(* CODESYS project Johnson,Joachim,Uppgift17.project

Project tree, tasks and I/O mapping:
  Device : CODESYS Control Win V3, 3S - Smart Software Solutions GmbH, order no. 305021, version 3.5.10.40
    application Application
      libraries: Standard, * (System)
      task MainTask (cyclic, interval t#20ms, priority 1) calls PLC_PRG, Lamp_Controll_Program [Controlling the lamp in the system], PrintoutAlarmCode
      program PLC_PRG [SFC]: MoveConv1to2, MoveCon2to3, Setrunning, SetStop, StopBTNCHECK, ResetAlarm, Convyor1to2Timout, Convyor2to3Timout
      global variables GVL
      Symbols
      program Lamp_Controll_Program [CFC]
      program Gui_Panel_Alarm [CFC]
      program PrintoutAlarmCode [CFC]
*)

// Device/Application/GVL
{attribute 'qualified_only'}
VAR_GLOBAL
	// signals from buttons
	iSUB00_S1: BOOL; // StartButton
	iSUB00_S2: BOOL; // Stopbutton
	iSUB00_S3: BOOL; // Resetbutton
	
	running: BOOL; 	// Is the aplication running
	alarm: BOOL; 	// Is the aplication running
	AlarmCode: word;
	
	// Signals from conveyors
	iSUB01_B1: BOOL; // Signals för conveyor 1. ontop
	iSUB02_B1: BOOL; // Signals för conveyor 2. ontop
	iSUB03_B1: BOOL; // Signals för conveyor 3. ontop
	
	// conveyor signal ontop conveyro.
	oSUB00_H1: BOOL; // Auto-On light
	oSUB00_H2: BOOL; // Alarm light
	oSUB00_H3: WORD; // Pallräknare
	
	// Motors
	oSUB01_K1: BOOL; // MOTOR FÖR converoyr 1
	oSUB02_K1: BOOL; // MOTOR FÖR converoyr 2
	oSUB03_K1: BOOL; // MOTOR FÖR converoyr 3
END_VAR

// Device/Application/PLC_PRG
PROGRAM PLC_PRG
VAR	
	TON_0: TON;
	OutputTime: TIME;
	TON2: TON;
	Output: TIME;
	TimeOutTimer: TON;
	TimeOutOutputTime: TIME;
	R_TRIG_0: R_TRIG;
	countercunt: CTD;
	countercunt3: CTD;
	countercunt4: CTD;
	Alarmcode: CTU;
	countercunt5: CTD;
END_VAR
VAR // added by the converter: edge detectors and wires of the graphical bodies
    _w1, _w3, _w5, _w6, _w12, _w14, _w15, _w17, _w19 : BOOL;
    _w2, _w4, _w7, _w8, _w9, _w10, _w11, _w13, _w16, _w18, _w20 : ANY;
END_VAR

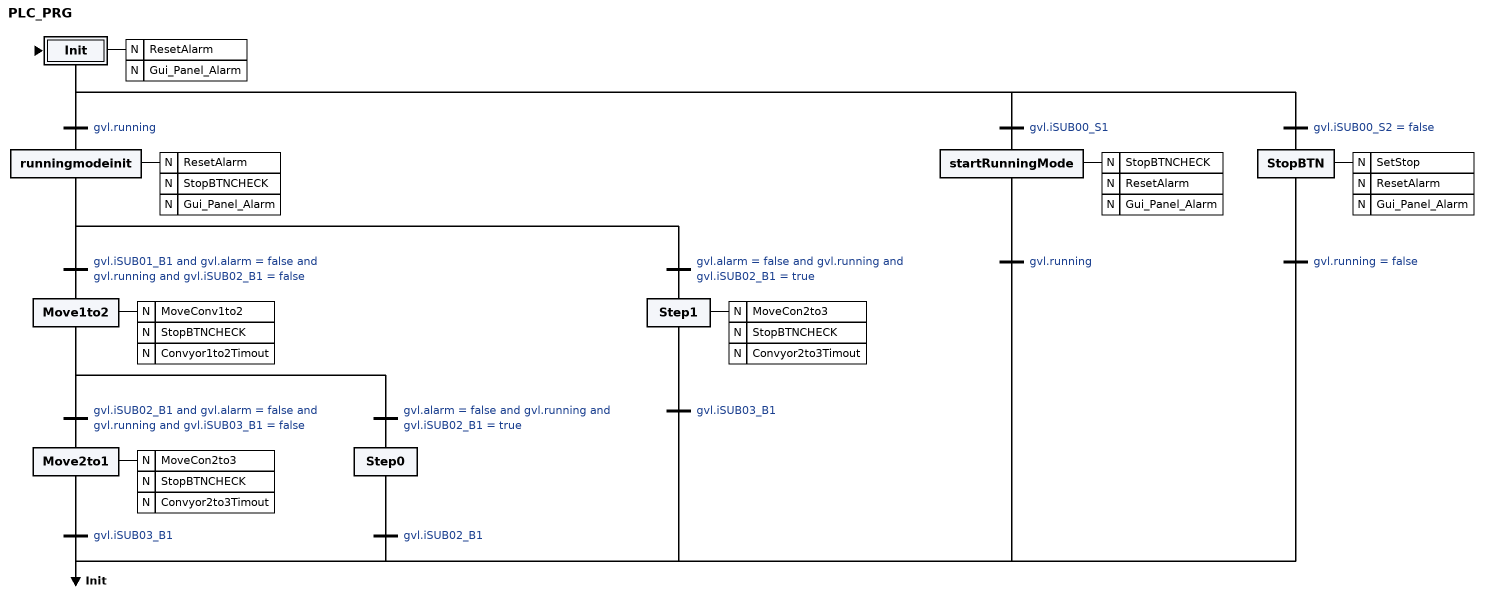
INITIAL_STEP Init:
    ResetAlarm(N);
    Gui_Panel_Alarm(N);
END_STEP
TRANSITION FROM Init TO runningmodeinit
    := gvl.running;
END_TRANSITION
STEP runningmodeinit:
    ResetAlarm(N);
    StopBTNCHECK(N);
    Gui_Panel_Alarm(N);
END_STEP
TRANSITION FROM runningmodeinit TO Move1to2
    := gvl.iSUB01_B1 and gvl.alarm = false and gvl.running and gvl.iSUB02_B1 = false;
END_TRANSITION
STEP Move1to2:
    MoveConv1to2(N);
    StopBTNCHECK(N);
    Convyor1to2Timout(N);
END_STEP
TRANSITION FROM Move1to2 TO Move2to1
    := gvl.iSUB02_B1 and gvl.alarm = false and gvl.running and gvl.iSUB03_B1 = false;
END_TRANSITION
STEP Move2to1:
    MoveCon2to3(N);
    StopBTNCHECK(N);
    Convyor2to3Timout(N);
END_STEP
TRANSITION FROM Move2to1 TO Init
    := gvl.iSUB03_B1;
END_TRANSITION
TRANSITION FROM Move1to2 TO Step0
    := gvl.alarm = false and gvl.running and gvl.iSUB02_B1 = true;
END_TRANSITION
STEP Step0:
END_STEP
TRANSITION FROM Step0 TO Init
    := gvl.iSUB02_B1;
END_TRANSITION
TRANSITION FROM runningmodeinit TO Step1
    := gvl.alarm = false and gvl.running and gvl.iSUB02_B1 = true;
END_TRANSITION
STEP Step1:
    MoveCon2to3(N);
    StopBTNCHECK(N);
    Convyor2to3Timout(N);
END_STEP
TRANSITION FROM Step1 TO Init
    := gvl.iSUB03_B1;
END_TRANSITION
TRANSITION FROM Init TO startRunningMode
    := gvl.iSUB00_S1;
END_TRANSITION
STEP startRunningMode:
    StopBTNCHECK(N);
    ResetAlarm(N);
    Gui_Panel_Alarm(N);
END_STEP
TRANSITION FROM startRunningMode TO Init
    := gvl.running;
END_TRANSITION
TRANSITION FROM Init TO StopBTN
    := gvl.iSUB00_S2 = false;
END_TRANSITION
STEP StopBTN:
    SetStop(N);
    ResetAlarm(N);
    Gui_Panel_Alarm(N);
END_STEP
TRANSITION FROM StopBTN TO Init
    := gvl.running = false;
END_TRANSITION

ACTION MoveConv1to2:
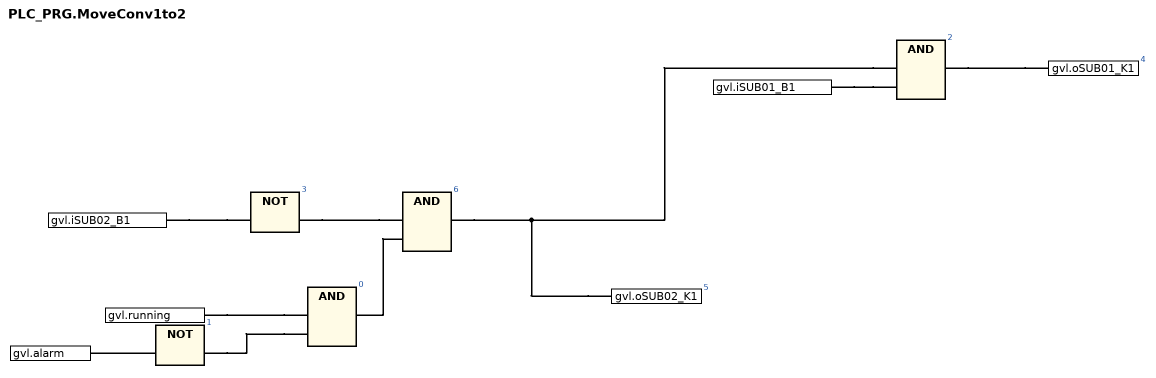
_w2 := gvl.running AND _w1;
_w1 := NOT gvl.alarm;
_w4 := NOT gvl.iSUB02_B1;
gvl.oSUB01_K1 := _w3 AND gvl.iSUB01_B1;
gvl.oSUB02_K1 := _w3;
_w3 := _w4 AND _w2;
END_ACTION

ACTION MoveCon2to3:
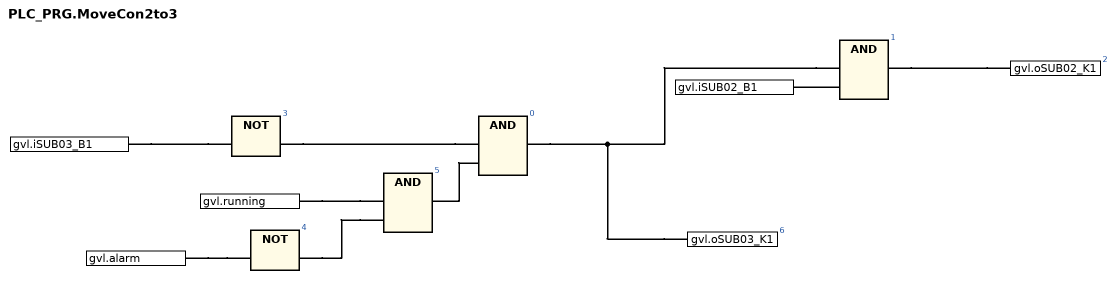
_w7 := _w5 AND _w6;
gvl.oSUB02_K1 := _w7 AND gvl.iSUB02_B1;
_w5 := NOT gvl.iSUB03_B1;
_w6 := gvl.running AND NOT gvl.alarm;
gvl.oSUB03_K1 := _w7;
END_ACTION

ACTION Setrunning:
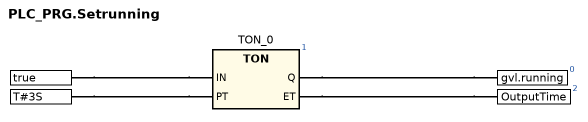
gvl.running := TON_0.Q;
TON_0(IN := true, PT := T#3S); // TON
OutputTime := TON_0.ET;
END_ACTION

ACTION SetStop:
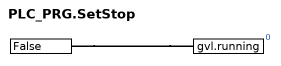
gvl.running := False;
END_ACTION

ACTION StopBTNCHECK:
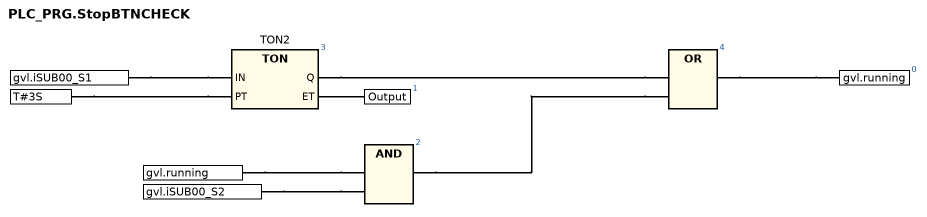
gvl.running := _w8;
Output := TON2.ET;
_w9 := gvl.running AND gvl.iSUB00_S2;
TON2(IN := gvl.iSUB00_S1, PT := T#3S); // TON
_w8 := TON2.Q OR _w9;
END_ACTION

ACTION ResetAlarm:
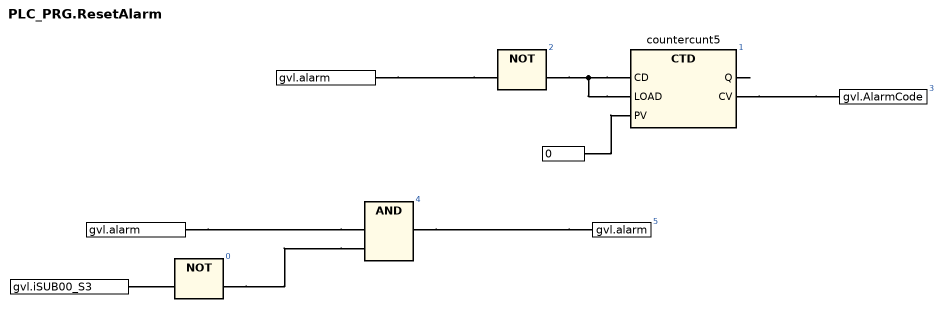
_w10 := NOT gvl.iSUB00_S3;
countercunt5(CD := _w11, LOAD := _w11, PV := 0); // CTD
_w11 := NOT gvl.alarm;
gvl.AlarmCode := countercunt5.CV;
gvl.alarm := gvl.alarm AND _w10;
END_ACTION

ACTION Convyor1to2Timout:
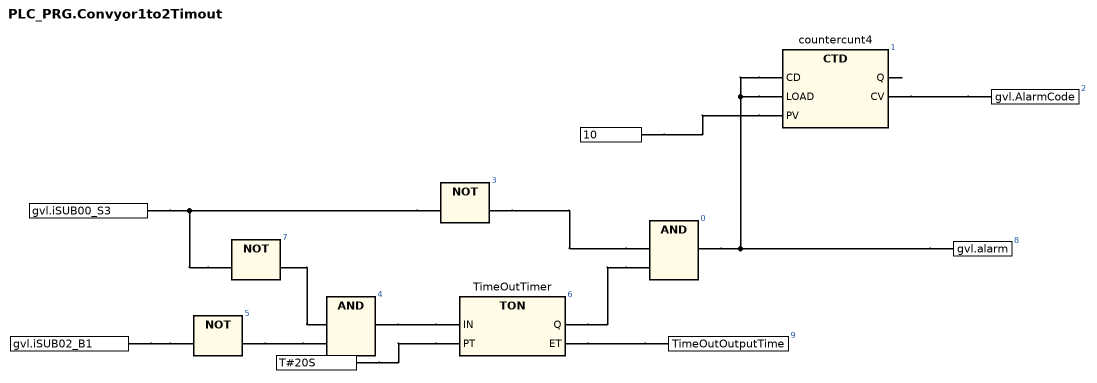
_w13 := _w12 AND TimeOutTimer.Q;
countercunt4(CD := _w13, LOAD := _w13, PV := 10); // CTD
gvl.AlarmCode := countercunt4.CV;
_w12 := NOT gvl.iSUB00_S3;
_w16 := _w14 AND _w15;
_w15 := NOT gvl.iSUB02_B1;
TimeOutTimer(IN := _w16, PT := T#20S); // TON
_w14 := NOT gvl.iSUB00_S3;
gvl.alarm := _w13;
TimeOutOutputTime := TimeOutTimer.ET;
END_ACTION

ACTION Convyor2to3Timout:
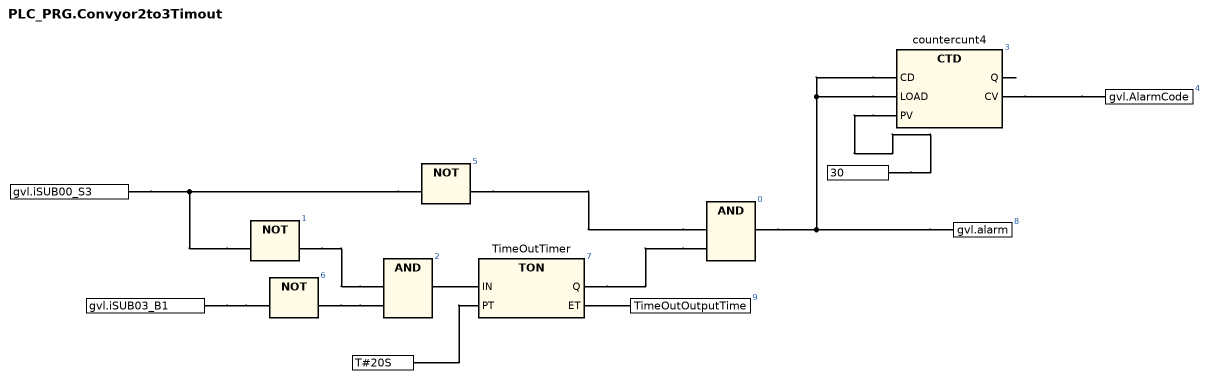
_w18 := _w17 AND TimeOutTimer.Q;
_w20 := NOT gvl.iSUB00_S3 AND _w19;
countercunt4(CD := _w18, LOAD := _w18, PV := 30); // CTD
gvl.AlarmCode := countercunt4.CV;
_w17 := NOT gvl.iSUB00_S3;
_w19 := NOT gvl.iSUB03_B1;
TimeOutTimer(IN := _w20, PT := T#20S); // TON
gvl.alarm := _w18;
TimeOutOutputTime := TimeOutTimer.ET;
END_ACTION

END_PROGRAM

// Device/Application/Lamp_Controll_Program
PROGRAM Lamp_Controll_Program
VAR
	Button_ON: TON;
	Button_Light_Off: TOF;
	Light_Time_TurnOff_Delay: TON;
	TurnLightOnTimeoutput: TIME;
	TurnLightOffTimeoutput: TIME;
END_VAR
VAR // added by the converter: edge detectors and wires of the graphical bodies
    _w1 : ANY;
    _w2 : BOOL;
END_VAR

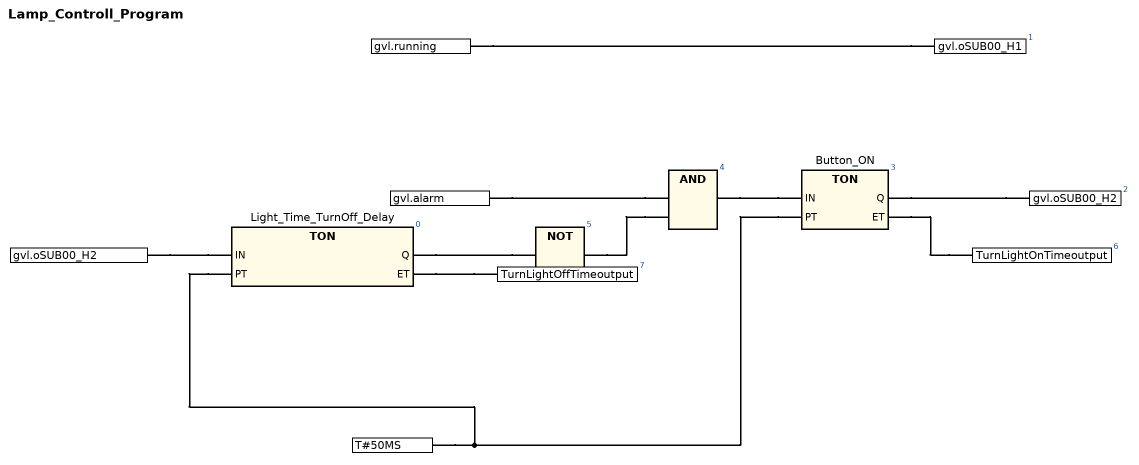
Light_Time_TurnOff_Delay(IN := gvl.oSUB00_H2, PT := T#50MS); // TON
gvl.oSUB00_H1 := gvl.running;
gvl.oSUB00_H2 := Button_ON.Q;
Button_ON(IN := _w1, PT := T#50MS); // TON
_w1 := gvl.alarm AND _w2;
_w2 := NOT Light_Time_TurnOff_Delay.Q;
TurnLightOnTimeoutput := Button_ON.ET;
TurnLightOffTimeoutput := Light_Time_TurnOff_Delay.ET;

END_PROGRAM

// Device/Application/PrintoutAlarmCode
PROGRAM PrintoutAlarmCode
VAR
END_VAR

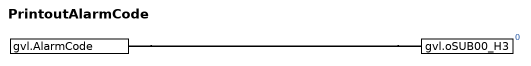
gvl.oSUB00_H3 := gvl.AlarmCode;

END_PROGRAM

// Device/Application/Gui_Panel_Alarm
PROGRAM Gui_Panel_Alarm
VAR
	TimeToAlarm: TON;
	TimeToAlarmOutput: TIME;
	countercunt2: CTD;
END_VAR
VAR // added by the converter: edge detectors and wires of the graphical bodies
    _w1, _w2, _w3 : ANY;
END_VAR

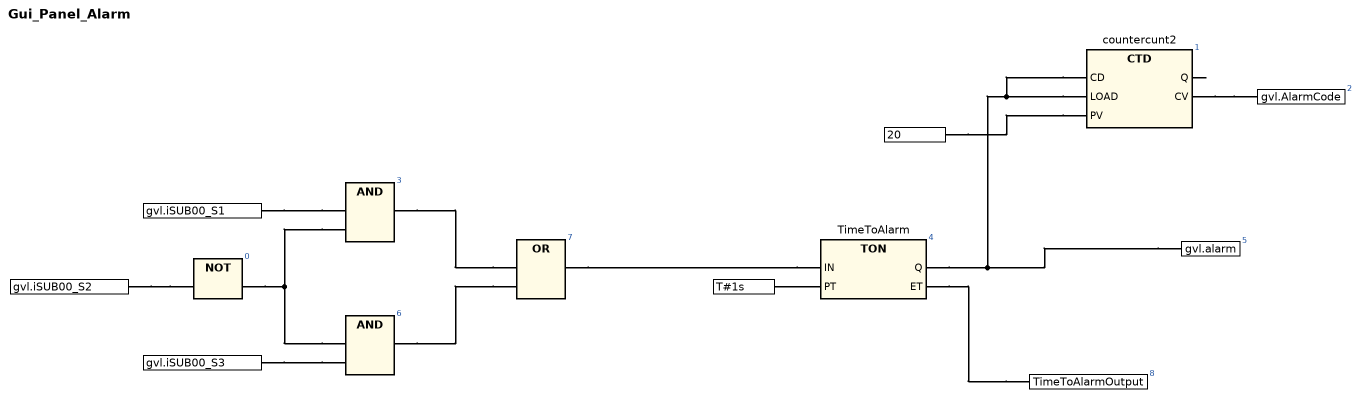
_w1 := NOT gvl.iSUB00_S2;
countercunt2(CD := TimeToAlarm.Q, LOAD := TimeToAlarm.Q, PV := 20); // CTD
gvl.AlarmCode := countercunt2.CV;
_w2 := gvl.iSUB00_S1 AND _w1;
TimeToAlarm(IN := _w3, PT := T#1s); // TON
gvl.alarm := TimeToAlarm.Q;
_w3 := _w2 OR _w1 AND gvl.iSUB00_S3;
TimeToAlarmOutput := TimeToAlarm.ET;

END_PROGRAM
